// TIA Portal V16 export
// export: Created 2022-02-28T20:45:44.416275Z, ExportSetting WithDefaults, DisplayName Totally Integrated Automation Portal, DisplayVersion V16, DisplayName TIA Portal Version Control Interface, DisplayVersion V16, DisplayName TIA Portal Openness, DisplayVersion V16, DisplayName STEP 7 Professional, DisplayVersion V16, DisplayName STEP 7 Safety, DisplayVersion V16, DisplayName WinCC Advanced, DisplayVersion V16
FUNCTION "02_Mapeo_Salida" : Void   // FC2, LAD
{ S7_Optimized_Access := 'TRUE' }
VERSION : 0.1
// stored: AutoNumber true, IsIECCheckEnabled false, SetENOAutomatically false, UDAEnableTagReadback false
BEGIN

REGION Network 1: Salidas Pistilos
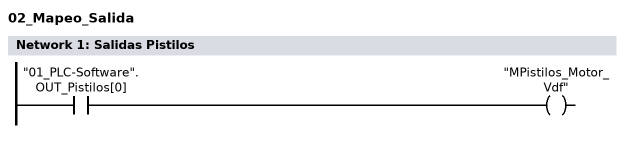
   RUNG wire#powerrail
      Contact( "01_PLC-Software".OUT_Pistilos[0] )
      Coil( "MPistilos_Motor_Vdf" )
   END_RUNG
   // the same network as SCL:
   "MPistilos_Motor_Vdf" := "01_PLC-Software".OUT_Pistilos[0];
END_REGION
END_FUNCTION
